{attribute 'qualified_only'}
VAR_GLOBAL
	nSample AT %I* : BOOL;
END_VAR

(* stored: Version 1.1.0.1, ProductVersion 3.1.4024.16
   GVL GVL_IO: Id {c60d839f-aaf4-4c67-aadf-e5e51c1108b8} *)
